// TIA Portal V18 export
DATA_BLOCK "Data"   // DB2
{ S7_Optimized_Access := 'FALSE' }
VERSION : 0.1
// stored: AutoNumber true, DBAccessibleFromOPCUA true, DBAccessibleFromWebserver true, IsOnlyStoredInLoadMemory false, IsWriteProtectedInAS false
   VAR
      steps_main : Int;
      steps_BoxCoveyor : Int;
      steps_Robot : Int;
      steps_PelletCoveyor : Int;
      steps_Storer : Int;
      last_step_BoxCoveyor : Int := 1;
      last_step_Robot : Int := 1;
      last_step_PalletCoveyor : Int := 1;
      last_step_Storer : Int := 1;
      status_box_movement : Bool := false;
      status_robot_movement : Bool := false;
      status_pallet_movement : Bool := false;
      status_capacitive_ready : Bool := false;
      status_storer_movement : Bool;
      fifo_boxes : "udt_Fifo";
      flanks : Array[0..31] of Bool;
      timers : Array[0..7] of TON_TIME;
      time_trigers : Array[0..7] of Bool;
   END_VAR
BEGIN
   fifo_boxes.Entrada.longitud := 31;
END_DATA_BLOCK
